// TIA Portal project "uygulama_2" (V18)

(* hardware
DEVICE "S7-1200 station_1"  S7-1200 Station
   slot 0: "Rack_0"  S7-1200 Rack  Rack  V1.0
   slot 1: "PLC_1"  CPU 1214C DC/DC/DC  6ES7 214-1AG40-0XB0  V4.6
*)

// ===== PLC "PLC_1"  CPU 1214C DC/DC/DC =====

VAR_GLOBAL   // PLC tag table "Default tag table"
   "STOP" AT %I0.0 : Bool;
   "START" AT %I0.1 : Bool;
   "1.MOTOR" AT %Q0.0 : Bool;
   "2.MOTOR" AT %Q0.1 : Bool;
   "YARDIMCI KONTAK" AT %M0.0 : Bool;
END_VAR

// folder: System blocks/Program resources

DATA_BLOCK "T1"   // DB1
{ S7_Optimized_Access := 'TRUE' }
AUTHOR : Simatic
FAMILY : IEC
NAME : IEC_TMR
VERSION : 1.0
// stored: InstanceOfName IEC_TIMER
"IEC_TIMER"
BEGIN
END_DATA_BLOCK

DATA_BLOCK "T2"   // DB2
{ S7_Optimized_Access := 'TRUE' }
AUTHOR : Simatic
FAMILY : IEC
NAME : IEC_TMR
VERSION : 1.0
// stored: InstanceOfName IEC_TIMER
"IEC_TIMER"
BEGIN
END_DATA_BLOCK

// folder: (top level)

ORGANIZATION_BLOCK "Main"   // OB1, LAD, ProgramCycle
TITLE = "Main Program Sweep (Cycle)"
{ S7_Optimized_Access := 'TRUE' }
VERSION : 0.1
   VAR_INPUT
      Initial_Call : Bool;   // Initial call of this OB
      Remanence : Bool;   // =True, if remanent data are available
   END_VAR
BEGIN

REGION Network 1
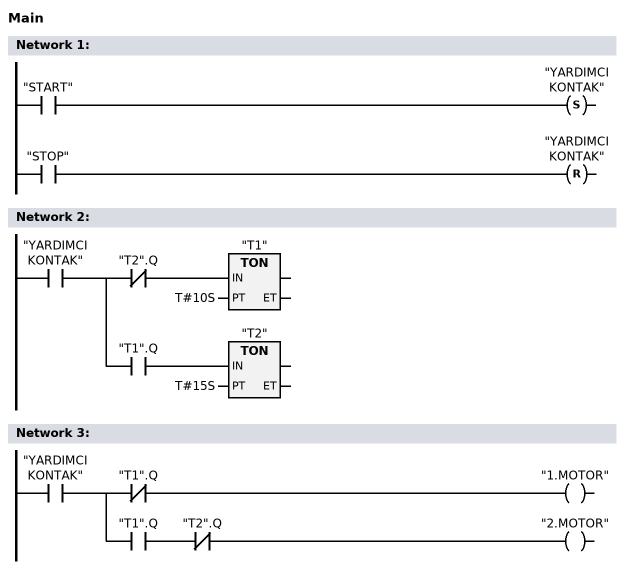
   RUNG wire#powerrail
      Contact( "START" )
      S_Coil( "YARDIMCI KONTAK" )
   END_RUNG
   RUNG wire#powerrail
      Contact( "STOP" )
      R_Coil( "YARDIMCI KONTAK" )
   END_RUNG
   // the same network as SCL:
   IF "START" THEN "YARDIMCI KONTAK" := TRUE; END_IF;
   IF "STOP" THEN "YARDIMCI KONTAK" := FALSE; END_IF;
END_REGION

REGION Network 2
   "T1".TON(IN := "YARDIMCI KONTAK" AND NOT "T2".Q, PT := T#10S);
   "T2".TON(IN := "YARDIMCI KONTAK" AND "T1".Q, PT := T#15S);
END_REGION

REGION Network 3
   RUNG wire#powerrail
      Contact( "YARDIMCI KONTAK" )
      wire#w1
      I_Contact( "T1".Q )
      Coil( "1.MOTOR" )
   END_RUNG
   RUNG wire#w1
      Contact( "T1".Q )
      I_Contact( "T2".Q )
      Coil( "2.MOTOR" )
   END_RUNG
   // the same network as SCL:
   "1.MOTOR" := "YARDIMCI KONTAK" AND NOT "T1".Q;
   "2.MOTOR" := "YARDIMCI KONTAK" AND "T1".Q AND NOT "T2".Q;
END_REGION
END_ORGANIZATION_BLOCK